INTERFACE IXtsHardware EXTENDS ICyclic

METHOD getAllMoversValid : BOOL
VAR_INPUT
END_VAR
END_METHOD

METHOD GetMoverEnvInterface : I_TcIoXtsXpuMover
VAR_INPUT
	MoverNumber : UINT;
END_VAR
END_METHOD

METHOD getMoversDetected : BOOL
VAR_INPUT
END_VAR
END_METHOD

METHOD IsInSim : BOOL
VAR_INPUT
END_VAR
END_METHOD

METHOD SetTracksForDetection : BOOL
VAR_INPUT
END_VAR
END_METHOD

METHOD TriggerMoverDetection : BOOL
VAR_INPUT
END_VAR
END_METHOD

METHOD TriggerMoverID : BOOL
VAR_INPUT
END_VAR
END_METHOD

END_INTERFACE

(* stored: Version 1.1.0.1, ProductVersion 3.1.4024.12
   Itf IXtsHardware: Id {bf384176-1154-4b20-87d2-6228ca722bc7}
   Method getAllMoversValid: Id {83cea3eb-034b-4ef6-97c8-3638f795443f}
   Method GetMoverEnvInterface: Id {06175234-441e-45a7-b310-01adbe58b90a}
   Method getMoversDetected: Id {b4027da9-aa3d-4e00-88aa-a047a5bd3219}
   Method IsInSim: Id {11de75bc-4a14-49be-839d-5d91f6e50bb8}
   Method SetTracksForDetection: Id {d824a2fc-c3a9-4504-ba47-b5bf353698b2}
   Method TriggerMoverDetection: Id {9ce51524-ddc5-4cb3-83bd-732953c72724}
   Method TriggerMoverID: Id {da9671e9-7f18-4b2b-82f9-ced25dd3dcd5} *)
